% RSLogix 500 project PROJECT4.RSS, saved by version 8.30.00.16 %
PROJECT "PROJECT4"    % processor: Bul.1763 MicroLogix 1100 Series B %

PROGRAM FILES
  LAD 2 "MAIN"  4 rungs
  LAD 3 "DI/DO"  7 rungs
  LAD 4 "CONTROL"  6 rungs
  LAD 5 "POSITION"  6 rungs

DATA FILES
  O0 OUTPUT  5 elements
  I1 INPUT  7 elements
  S2 STATUS  66 elements
  B3 BINARY  1 elements
  T4 TIMER  3 elements
  C5 COUNTER  1 elements
  R6 CONTROL  1 elements
  N7 INTEGER  1 elements
  F8 FLOAT  1 elements

LADDER 2 "MAIN"
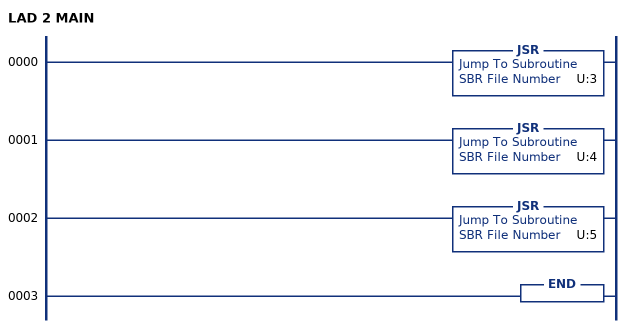
% Rung: 0 %
SOR JSR U:3 EOR
% Rung: 1 %
SOR JSR U:4 EOR
% Rung: 2 %
SOR JSR U:5 EOR
% Rung: 3 %
SOR END EOR

LADDER 3 "DI/DO"
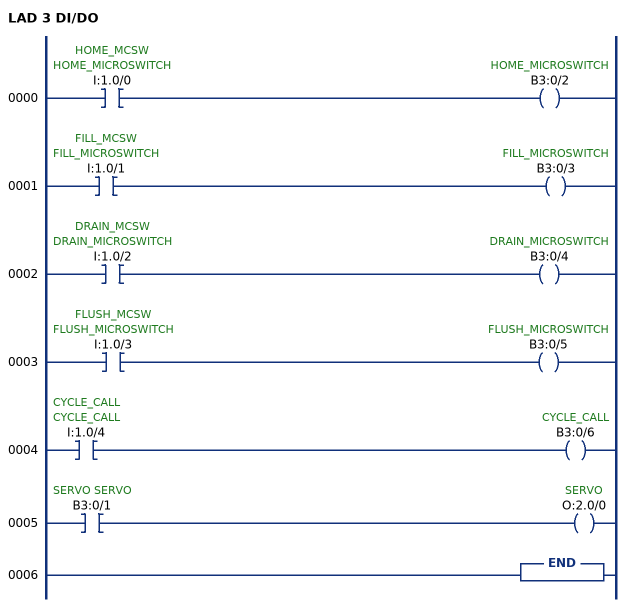
% Rung: 0 %
SOR XIC I:1.0/0 OTE B3:0/2 EOR
%   I:1.0/0  HOME_MICROSWITCH  "HOME_MCSW" %
%   B3:0/2  "HOME_MICROSWITCH" %
% Rung: 1 %
SOR XIC I:1.0/1 OTE B3:0/3 EOR
%   I:1.0/1  FILL_MICROSWITCH  "FILL_MCSW" %
%   B3:0/3  "FILL_MICROSWITCH" %
% Rung: 2 %
SOR XIC I:1.0/2 OTE B3:0/4 EOR
%   I:1.0/2  DRAIN_MICROSWITCH  "DRAIN_MCSW" %
%   B3:0/4  "DRAIN_MICROSWITCH" %
% Rung: 3 %
SOR XIC I:1.0/3 OTE B3:0/5 EOR
%   I:1.0/3  FLUSH_MICROSWITCH  "FLUSH_MCSW" %
%   B3:0/5  "FLUSH_MICROSWITCH" %
% Rung: 4 %
SOR XIC I:1.0/4 OTE B3:0/6 EOR
%   I:1.0/4  CYCLE_CALL  "CYCLE_CALL" %
%   B3:0/6  "CYCLE_CALL" %
% Rung: 5 %
SOR XIC B3:0/1 OTE O:2.0/0 EOR
%   B3:0/1  SERVO  "SERVO" %
%   O:2.0/0  "SERVO" %
% Rung: 6 %
SOR END EOR

LADDER 4 "CONTROL"
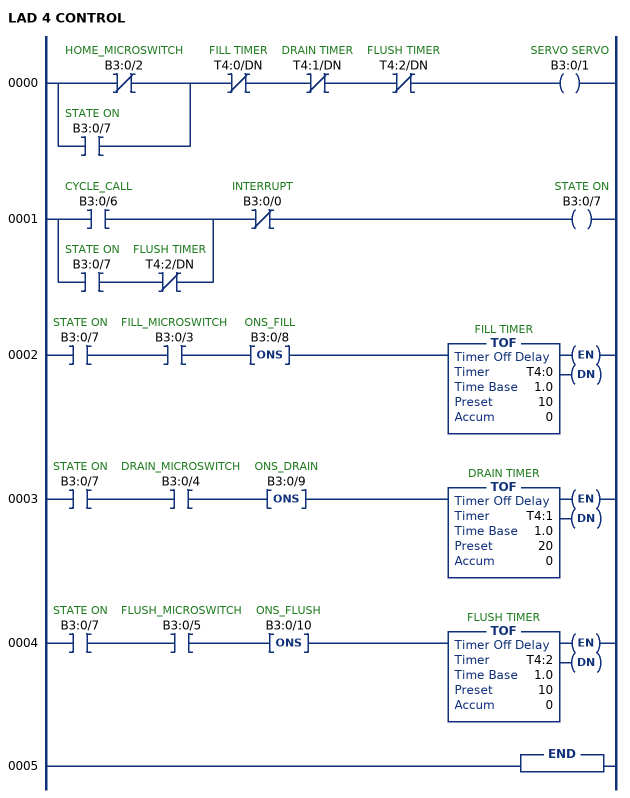
% Rung: 0 %
SOR BST XIO B3:0/2 NXB XIC B3:0/7 BND XIO T4:0/DN XIO T4:1/DN XIO T4:2/DN OTE B3:0/1 EOR
%   B3:0/2  "HOME_MICROSWITCH" %
%   B3:0/7  "STATE ON" %
%   T4:0  "FILL TIMER" %
%   T4:1  "DRAIN TIMER" %
%   T4:2  "FLUSH TIMER" %
%   B3:0/1  SERVO  "SERVO" %
% Rung: 1 %
SOR BST XIC B3:0/6 NXB XIC B3:0/7 XIO T4:2/DN BND XIO B3:0/0 OTE B3:0/7 EOR
%   B3:0/6  "CYCLE_CALL" %
%   B3:0/7  "STATE ON" %
%   T4:2  "FLUSH TIMER" %
%   B3:0/0  "INTERRUPT" %
% Rung: 2 %
SOR XIC B3:0/7 XIC B3:0/3 ONS B3:0/8 TOF T4:0 1.0 10 0 EOR
%   B3:0/7  "STATE ON" %
%   B3:0/3  "FILL_MICROSWITCH" %
%   B3:0/8  "ONS_FILL" %
%   T4:0  "FILL TIMER" %
% Rung: 3 %
SOR XIC B3:0/7 XIC B3:0/4 ONS B3:0/9 TOF T4:1 1.0 20 0 EOR
%   B3:0/7  "STATE ON" %
%   B3:0/4  "DRAIN_MICROSWITCH" %
%   B3:0/9  "ONS_DRAIN" %
%   T4:1  "DRAIN TIMER" %
% Rung: 4 %
SOR XIC B3:0/7 XIC B3:0/5 ONS B3:0/10 TOF T4:2 1.0 10 0 EOR
%   B3:0/7  "STATE ON" %
%   B3:0/5  "FLUSH_MICROSWITCH" %
%   B3:0/10  "ONS_FLUSH" %
%   T4:2  "FLUSH TIMER" %
% Rung: 5 %
SOR END EOR

LADDER 5 "POSITION"
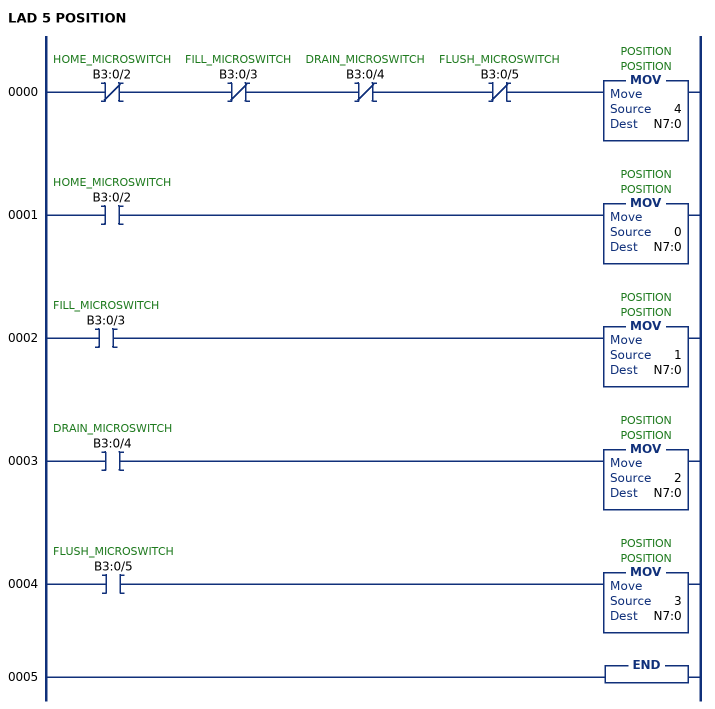
% Rung: 0 %
SOR XIO B3:0/2 XIO B3:0/3 XIO B3:0/4 XIO B3:0/5 MOV 4 N7:0 EOR
%   B3:0/2  "HOME_MICROSWITCH" %
%   B3:0/3  "FILL_MICROSWITCH" %
%   B3:0/4  "DRAIN_MICROSWITCH" %
%   B3:0/5  "FLUSH_MICROSWITCH" %
%   N7:0  POSITION  "POSITION" %
% Rung: 1 %
SOR XIC B3:0/2 MOV 0 N7:0 EOR
%   B3:0/2  "HOME_MICROSWITCH" %
%   N7:0  POSITION  "POSITION" %
% Rung: 2 %
SOR XIC B3:0/3 MOV 1 N7:0 EOR
%   B3:0/3  "FILL_MICROSWITCH" %
%   N7:0  POSITION  "POSITION" %
% Rung: 3 %
SOR XIC B3:0/4 MOV 2 N7:0 EOR
%   B3:0/4  "DRAIN_MICROSWITCH" %
%   N7:0  POSITION  "POSITION" %
% Rung: 4 %
SOR XIC B3:0/5 MOV 3 N7:0 EOR
%   B3:0/5  "FLUSH_MICROSWITCH" %
%   N7:0  POSITION  "POSITION" %
% Rung: 5 %
SOR END EOR

DATA TABLE (non-zero values as saved)
DATA T4
% .PRE .ACC %
% T4:0 % 10 0
% T4:1 % 20 0
% T4:2 % 10 0
